Yaskawa INFORM job: kufsa_test.JBI

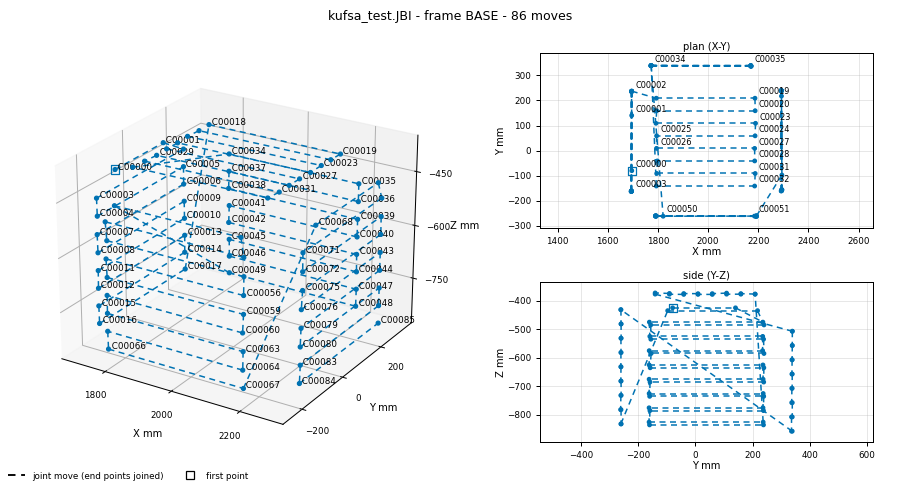
[picture p0: tool path of kufsa_test.JBI in frame BASE, 86 of 86 moves have a stored position in this frame; points joined in program order, loops and branches not executed]
/JOB
//NAME kufsa_test
//POS
///NPOS 86,0,0,0,0,0
///TOOL 0
///POSTYPE BASE
///RECTAN
///RCONF 1,0,0,0,0,0,0,0,0,0,0,0,0,0,0,0,0,0,0,0,0,0,0,0
C00000=1696.132,-80.047,-425.128,0.0000,90.0000,0.0000
C00001=1695.649,140.027,-425.128,0.0000,90.0000,0.0000
C00002=1695.009,236.007,-475.128,0.0000,90.0000,0.0000
C00003=1694.894,-161.509,-475.128,0.0000,90.0000,0.0000
C00004=1694.500,-159.876,-525.128,0.0000,90.0000,0.0000
C00005=1694.957,235.269,-525.128,0.0000,90.0000,0.0000
C00006=1695.172,234.870,-575.128,0.0000,90.0000,0.0000
C00007=1694.072,-162.036,-575.128,0.0000,90.0000,0.0000
C00008=1695.266,-162.303,-625.128,0.0000,90.0000,0.0000
C00009=1695.465,236.123,-625.128,0.0000,90.0000,0.0000
C00010=1695.422,236.644,-675.128,0.0000,90.0000,0.0000
C00011=1694.457,-162.352,-675.128,0.0000,90.0000,0.0000
C00012=1693.613,-162.296,-725.128,0.0000,90.0000,0.0000
C00013=1695.359,236.966,-725.128,0.0000,90.0000,0.0000
C00014=1695.305,236.328,-775.128,0.0000,90.0000,0.0000
C00015=1693.299,-162.503,-775.128,0.0000,90.0000,0.0000
C00016=1694.079,-162.510,-825.128,0.0000,90.0000,0.0000
C00017=1695.793,236.889,-825.128,0.0000,90.0000,0.0000
C00018=1793.675,208.803,-377.180,-180.0000,0.0000,90.0000
C00019=2187.017,208.803,-377.015,-180.0000,0.0000,90.0000
C00020=2187.698,158.803,-375.418,-180.0000,0.0000,90.0000
C00021=1795.170,158.803,-377.409,-180.0000,0.0000,90.0000
C00022=1792.375,108.803,-377.337,-180.0000,0.0000,90.0000
C00023=2189.165,108.803,-373.615,-180.0000,0.0000,90.0000
C00024=2187.408,58.803,-375.476,-180.0000,0.0000,90.0000
C00025=1795.003,58.803,-378.201,-180.0000,0.0000,90.0000
C00026=1794.543,8.803,-378.074,-180.0000,0.0000,90.0000
C00027=2185.685,8.803,-375.544,-180.0000,0.0000,90.0000
C00028=2185.880,-41.196,-375.195,-180.0000,0.0000,90.0000
C00029=1797.809,-41.196,-378.167,-180.0000,0.0000,90.0000
C00030=1795.305,-91.196,-377.541,-180.0000,0.0000,90.0000
C00031=2187.800,-91.196,-374.817,-180.0000,0.0000,90.0000
C00032=2185.655,-141.196,-373.016,-180.0000,0.0000,90.0000
C00033=1793.794,-141.196,-377.211,-180.0000,0.0000,90.0000
C00034=1773.422,338.858,-507.069,90.0000,0.0000,0.0000
C00035=2170.526,339.076,-507.069,90.0000,0.0000,0.0000
C00036=2170.470,338.721,-557.069,90.0000,0.0000,0.0000
C00037=1772.765,338.845,-557.069,90.0000,0.0000,0.0000
C00038=1772.113,338.178,-607.069,90.0000,0.0000,0.0000
C00039=2169.918,338.249,-607.069,90.0000,0.0000,0.0000
C00040=2169.846,337.617,-657.069,90.0000,0.0000,0.0000
C00041=1773.408,338.699,-657.069,90.0000,0.0000,0.0000
C00042=1771.966,338.269,-707.069,90.0000,0.0000,0.0000
C00043=2169.887,337.437,-707.069,90.0000,0.0000,0.0000
C00044=2170.816,336.900,-757.069,90.0000,0.0000,0.0000
C00045=1773.075,338.832,-757.069,90.0000,0.0000,0.0000
C00046=1773.335,338.792,-807.069,90.0000,0.0000,0.0000
C00047=2171.727,336.247,-807.069,90.0000,0.0000,0.0000
C00048=2171.220,336.110,-857.069,90.0000,0.0000,0.0000
C00049=1773.221,338.627,-857.069,90.0000,0.0000,0.0000
C00050=1820.971,-261.541,-431.614,-90.0000,0.0000,0.0000
C00051=2184.952,-261.044,-431.614,-90.0000,0.0000,0.0000
C00052=2192.839,-260.681,-481.614,-90.0000,0.0000,0.0000
C00053=1791.152,-260.567,-481.614,0.0000,90.0000,0.0000
C00054=1794.425,-260.324,-531.614,-90.0000,0.0000,0.0000
C00055=2193.314,-261.064,-531.614,-90.0000,0.0000,0.0000
C00056=2192.341,-260.734,-581.614,-90.0000,0.0000,0.0000
C00057=1791.071,-261.005,-581.614,-90.0000,0.0000,0.0000
C00058=1793.131,-261.280,-631.614,-90.0000,0.0000,0.0000
C00059=2192.209,-260.873,-631.614,-90.0000,0.0000,0.0000
C00060=2189.954,-261.359,-681.614,-90.0000,0.0000,0.0000
C00061=1791.050,-260.611,-681.614,-90.0000,0.0000,0.0000
C00062=1790.464,-260.376,-731.614,-90.0000,0.0000,0.0000
C00063=2191.354,-261.246,-731.614,-90.0000,0.0000,0.0000
C00064=2190.798,-262.036,-781.614,-90.0000,0.0000,0.0000
C00065=1790.058,-260.739,-781.614,-90.0000,0.0000,0.0000
C00066=1790.686,-260.189,-831.614,-90.0000,0.0000,0.0000
C00067=2192.318,-261.278,-831.614,-90.0000,0.0000,0.0000
C00068=2294.292,-97.327,-435.033,0.0000,0.0000,0.0000
C00069=2292.553,217.265,-435.033,0.0000,0.0000,0.0000
C00070=2291.804,239.786,-485.033,0.0000,0.0000,0.0000
C00071=2294.201,-156.615,-485.033,0.0000,0.0000,0.0000
C00072=2293.933,-156.359,-535.033,0.0000,0.0000,0.0000
C00073=2292.245,238.334,-535.033,0.0000,0.0000,0.0000
C00074=2291.848,239.682,-585.033,0.0000,0.0000,0.0000
C00075=2293.799,-155.333,-585.033,0.0000,0.0000,0.0000
C00076=2292.833,-158.703,-635.033,0.0000,0.0000,0.0000
C00077=2291.947,239.284,-635.033,0.0000,0.0000,0.0000
C00078=2292.084,238.852,-685.033,0.0000,0.0000,0.0000
C00079=2292.973,-159.159,-685.033,0.0000,0.0000,0.0000
C00080=2292.114,-160.465,-735.033,0.0000,0.0000,0.0000
C00081=2291.977,238.820,-735.033,0.0000,0.0000,0.0000
C00082=2292.135,237.997,-785.033,0.0000,0.0000,0.0000
C00083=2292.381,-159.627,-785.033,0.0000,0.0000,0.0000
C00084=2291.307,-160.899,-835.033,0.0000,0.0000,0.0000
C00085=2292.416,237.973,-835.033,0.0000,0.0000,0.0000
//INST
///DATE 2023/01/01 11:40
///ATTR SC,RW,RJ
////FRAME BASE
///GROUP1 RB1
NOP
MOVJ C00000 VJ=15.00
MOVJ C00001 VJ=15.00
MOVJ C00002 VJ=15.00
MOVJ C00003 VJ=15.00
MOVJ C00004 VJ=15.00
MOVJ C00005 VJ=15.00
MOVJ C00006 VJ=15.00
MOVJ C00007 VJ=15.00
MOVJ C00008 VJ=15.00
MOVJ C00009 VJ=15.00
MOVJ C00010 VJ=15.00
MOVJ C00011 VJ=15.00
MOVJ C00012 VJ=15.00
MOVJ C00013 VJ=15.00
MOVJ C00014 VJ=15.00
MOVJ C00015 VJ=15.00
MOVJ C00016 VJ=15.00
MOVJ C00017 VJ=15.00
MOVJ C00018 VJ=15.00
MOVJ C00019 VJ=15.00
MOVJ C00020 VJ=15.00
MOVJ C00021 VJ=15.00
MOVJ C00022 VJ=15.00
MOVJ C00023 VJ=15.00
MOVJ C00024 VJ=15.00
MOVJ C00025 VJ=15.00
MOVJ C00026 VJ=15.00
MOVJ C00027 VJ=15.00
MOVJ C00028 VJ=15.00
MOVJ C00029 VJ=15.00
MOVJ C00030 VJ=15.00
MOVJ C00031 VJ=15.00
MOVJ C00032 VJ=15.00
MOVJ C00033 VJ=15.00
MOVJ C00034 VJ=15.00
MOVJ C00035 VJ=15.00
MOVJ C00036 VJ=15.00
MOVJ C00037 VJ=15.00
MOVJ C00038 VJ=15.00
MOVJ C00039 VJ=15.00
MOVJ C00040 VJ=15.00
MOVJ C00041 VJ=15.00
MOVJ C00042 VJ=15.00
MOVJ C00043 VJ=15.00
MOVJ C00044 VJ=15.00
MOVJ C00045 VJ=15.00
MOVJ C00046 VJ=15.00
MOVJ C00047 VJ=15.00
MOVJ C00048 VJ=15.00
MOVJ C00049 VJ=15.00
MOVJ C00050 VJ=15.00
MOVJ C00051 VJ=15.00
MOVJ C00052 VJ=15.00
MOVJ C00053 VJ=15.00
MOVJ C00054 VJ=15.00
MOVJ C00055 VJ=15.00
MOVJ C00056 VJ=15.00
MOVJ C00057 VJ=15.00
MOVJ C00058 VJ=15.00
MOVJ C00059 VJ=15.00
MOVJ C00060 VJ=15.00
MOVJ C00061 VJ=15.00
MOVJ C00062 VJ=15.00
MOVJ C00063 VJ=15.00
MOVJ C00064 VJ=15.00
MOVJ C00065 VJ=15.00
MOVJ C00066 VJ=15.00
MOVJ C00067 VJ=15.00
MOVJ C00068 VJ=15.00
MOVJ C00069 VJ=15.00
MOVJ C00070 VJ=15.00
MOVJ C00071 VJ=15.00
MOVJ C00072 VJ=15.00
MOVJ C00073 VJ=15.00
MOVJ C00074 VJ=15.00
MOVJ C00075 VJ=15.00
MOVJ C00076 VJ=15.00
MOVJ C00077 VJ=15.00
MOVJ C00078 VJ=15.00
MOVJ C00079 VJ=15.00
MOVJ C00080 VJ=15.00
MOVJ C00081 VJ=15.00
MOVJ C00082 VJ=15.00
MOVJ C00083 VJ=15.00
MOVJ C00084 VJ=15.00
MOVJ C00085 VJ=15.00
END
